PROGRAM P_HMI

VAR
    //bBlink : BOOL; // This variable toggles to create the blinking effect.
    tBlinkTimer : TON; // TON timer for controlling the blink rate.

	
	tSampleTimer: TON; // Timer for controlling the sampling rate
    nIndex: INT := 1; // Index for the next sample to be stored

END_VAR


HMI.bData1 := HMI.bP_PI; 
G_IO.P_Gain := HMI.bP_PI;

HMI.bDataP_DC := HMI.bProtielGainP_DC; 
HMI.bDataP_DC := HMI.bProtielGainP_DC; 


HMI.bData2 := HMI.bI_PI; 
G_IO.I_Gain := HMI.bI_PI;
// Enbiling the Ovrider fore END Stop //// 
/// HMI.bEndStopOverride := 

 

// Set the timer. It will start counting when IN is TRUE and reset when IN is FALSE.
tBlinkTimer(IN := NOT tBlinkTimer.Q, PT := T#1S); // The timer period is set to 1 second.

// Toggle the blink variable when the timer elapses (Q turns TRUE).
IF HMI.bEndStopOverride THEN
	IF tBlinkTimer.Q THEN
		HMI.bBlink := NOT HMI.bBlink;
	END_IF;
ELSE 
	HMI.bBlink := FALSE;
	
END_IF; 


IF HMI.bSwichForPlot THEN
	IF tBlinkTimer.Q THEN
		HMI.bSampleReady := NOT HMI.bSampleReady;
	END_IF;
ELSE 
	HMI.bSwichForPlot := FALSE;
	
END_IF; 


// for ploting the pistion of the system on vizualizer 
IF HMI.bSampleReady THEN
    HMI.arrPayLoadPositions[nIndex] := G_Sensors.fPayLoadPosition; // Store the current position
    
    nIndex := nIndex + 1; // Move to the next index
    IF nIndex > 100 THEN
        nIndex := 1; // Reset the index to create a circular buffer
    END_IF;
    
   HMI.bSampleReady := FALSE; // Reset the sample trigger
END_IF;


// for ploting the Sin Wave on vizualizer 
IF HMI.bSampleReady THEN
    HMI.arrSinPayLoadPositions[nIndex] := G_IO.SinuSignal; // Store the current position
    
    nIndex := nIndex + 1; // Move to the next index
    IF nIndex > 100 THEN
        nIndex := 1; // Reset the index to create a circular buffer
    END_IF;
    
   HMI.bSampleReady := FALSE; // Reset the sample trigger
END_IF;



IF HMI.bActvateSMC THEN
	IF tBlinkTimer.Q THEN
		HMI.bSampleReady := NOT HMI.bSampleReady;
	END_IF;
ELSE 
	HMI.bActvateSMC := FALSE;
	
END_IF; 


// for ploting the pistion of the system on vizualizer 
IF HMI.bSampleReady THEN
    HMI.arrPayLoadPositions[nIndex] := G_Sensors.fYokeNormalizedFeedback; // Store the current position
    
    nIndex := nIndex + 1; // Move to the next index
    IF nIndex > 100 THEN
        nIndex := 1; // Reset the index to create a circular buffer
    END_IF;
    
   HMI.bSampleReady := FALSE; // Reset the sample trigger
END_IF;

END_PROGRAM

(* stored: Version 1.1.0.1, ProductVersion 3.1.4024.12
   POU P_HMI: Id {bc7b7dbf-743d-4b40-85bd-31d52f5cea50}, SpecialFunc None *)
